// TIA Portal V18 export
// export: Created 2023-08-15T09:31:45.3155341Z, ExportSetting WithDefaults, DisplayName Totally Integrated Automation Portal, DisplayVersion V18 Update 2, DisplayName TIA Portal Openness, DisplayVersion V18 Update 2, DisplayName TIA Portal Version Control Interface, DisplayVersion V18, DisplayName SINAMICS Startdrive Advanced, DisplayVersion V18, DisplayName SINAMICS Startdrive G130, G150, S120, S150, SINAMICS MV, S210, DisplayVersion V18, DisplayName SINAMICS Startdrive G110M, G120, G120C, G120D, G120P, G115D, DisplayVersion V18, DisplayName STEP 7 Professional, DisplayVersion V18 Update 2, DisplayName STEP 7 Safety, DisplayVersion V18, DisplayName WinCC Advanced / Unified PC, DisplayVersion V18 Update 2
DATA_BLOCK "DrivesData"   // DB2
{ S7_Optimized_Access := 'TRUE' }
VERSION : 0.1
// stored: AutoNumber true, DBAccessibleFromOPCUA true, DBAccessibleFromWebserver true, IsOnlyStoredInLoadMemory false, IsRetainMemResEnabled false, IsWriteProtectedInAS false, MemoryReserve 100
   VAR
      kuljetin : "typeSinaSpeedInterface";
   END_VAR
BEGIN
   kuljetin.control.hwidStw := 266;
   kuljetin.control.hwidZsw := 266;
END_DATA_BLOCK
